{attribute 'linkalways'} 
{attribute 'no_explicit_call' := 'This FB is a CLASS and must be accessed using methods or properties'}
{attribute 'enable_dynamic_creation'}
FUNCTION_BLOCK _ETcWatchdogAccumulationType EXTENDS EnumDatatypeBase
VAR
	localData : ETcWatchdogAccumulationType;
	activeData : REFERENCE TO ETcWatchdogAccumulationType;
	enumBaseDatatype : _UINT(localData);
END_VAR

METHOD PRIVATE AddLocalEnumeration
VAR_INPUT
	Enumeration : T_MAXSTRING;
	Value : ETcWatchdogAccumulationType;
END_VAR
AddEnumeration(Enumeration, Value);
END_METHOD

PROPERTY PUBLIC Address : PVOID
GET
Address := ADR(activeData);
END_GET
END_PROPERTY

METHOD PUBLIC ClearReference
VAR_INPUT
END_VAR
activeData REF= localData;
SetBaseDatatypeReference();
END_METHOD

METHOD PUBLIC Clone : I_Datatype
VAR
    pClone : POINTER TO _ETcWatchdogAccumulationType;
END_VAR
pClone := __NEW(_ETcWatchdogAccumulationType(InitialValue := Value));
Clone := pClone^;
END_METHOD

METHOD FB_init : BOOL
VAR_INPUT
	bInitRetains : BOOL; // if TRUE, the retain variables are initialized (warm start / cold start)
	bInCopyCode : BOOL;  // if TRUE, the instance afterwards gets moved into the copy code (online change)
	InitialValue : ETcWatchdogAccumulationType;
END_VAR
localData := InitialValue;
AddBaseDatatype(enumBaseDatatype);
ClearReference();

AddLocalEnumeration('WD_ACC_TYPE_MEAN', ETcWatchdogAccumulationType.WD_ACC_TYPE_MEAN);
AddLocalEnumeration('WD_ACC_TYPE_PRODUCT', ETcWatchdogAccumulationType.WD_ACC_TYPE_PRODUCT);
END_METHOD

PROPERTY PUBLIC Identifier : T_MAXSTRING
GET
Identifier := 'ETcWatchdogAccumulationType';
END_GET
END_PROPERTY

METHOD IsEnumeratorValueEqual : BOOL
VAR_INPUT
	Enumerator : I_KeyValueForwardEnumerator;
END_VAR
VAR
	storedValue : ETcWatchdogAccumulationType;
END_VAR
IF NOT Enumerator.TryGet(storedValue) THEN
	RETURN;
END_IF

IsEnumeratorValueEqual := storedValue = activeData;
END_METHOD

METHOD PUBLIC MakeReferenceTo
VAR_INPUT
	ReferenceTarget : REFERENCE TO ETcWatchdogAccumulationType;
END_VAR
activeData REF= ReferenceTarget;
SetBaseDatatypeReference();
END_METHOD

METHOD PROTECTED SetBaseDatatypeReference
VAR_INPUT
END_VAR
enumBaseDatatype.MakeReferenceTo(activeData);
END_METHOD

PROPERTY PUBLIC Size : UDINT
GET
Size := SIZEOF(activeData);
END_GET
END_PROPERTY

METHOD TryMakeReferenceTo : BOOL
VAR_INPUT
	Target : I_Datatype;
END_VAR
VAR
	targetAsEnum : I_EnumDatatype;
	pTargetData : POINTER TO ETcWatchdogAccumulationType;
END_VAR
IF NOT Target.TryResolveAsEnumDatatype(targetAsEnum) THEN
	RETURN;
END_IF

IF targetAsEnum.Identifier <> Identifier THEN
	RETURN;
END_IF

pTargetData := Target.Address;
activeData REF= pTargetData^;
SetBaseDatatypeReference();
TryMakeReferenceTo := TRUE;
END_METHOD

PROPERTY PUBLIC Value : ETcWatchdogAccumulationType
GET
Value := activeData;
END_GET
SET
activeData := Value;
END_SET
END_PROPERTY

END_FUNCTION_BLOCK

(* stored: Version 1.1.0.1
   POU _ETcWatchdogAccumulationType: Id {9f8e712b-221d-4b7e-b23d-5a6a9598707e}, SpecialFunc None
   Folder Constructor: Id {27fa2eca-7872-442a-902d-23232a8fd823}
   Folder Private: Id {269bf6d6-2bb1-4317-9a0b-7ba3ebc69cf2}
   Folder Protected: Id {27d71b63-69c6-4680-925a-32c6207d271a}
   Method AddLocalEnumeration: Id {07002d06-a67f-4aba-b328-3283cf7e4720}
   Property Address: Id {1f239f12-6e32-4dcd-ab6c-6a0ce4ef1111}
   Get Get: Id {4769a909-79a9-470c-ae4f-3b56ce2ea6f9}
   Method ClearReference: Id {28bdb0ed-da8b-44d6-9f97-70731fff0c14}
   Method Clone: Id {6c808ac7-8fbb-4052-95bd-8df91069ec9b}
   Method FB_init: Id {634ef7f5-6f96-4ba5-b9a9-01fa2cf31a10}
   Property Identifier: Id {0ffe4e56-f1d2-4d1c-8de7-916a00535246}
   Get Get: Id {2633fb2b-a053-4228-b875-a7050c1535ff}
   Method IsEnumeratorValueEqual: Id {f02bc429-b086-42d4-b511-c7b98a1c12ff}
   Method MakeReferenceTo: Id {6e05ed69-6db9-4733-b551-c0c1f5e812dc}
   Method SetBaseDatatypeReference: Id {e6be49f2-20bf-4f80-ba26-a001d5b35436}
   Property Size: Id {19e13549-991c-4aa7-9d39-466cda80e336}
   Get Get: Id {bc022000-e4f6-4bae-8e46-482217014613}
   Method TryMakeReferenceTo: Id {12b1ec98-d1e3-48e8-b968-f53f969e7356}
   Property Value: Id {34a5055c-b9da-4aa6-8f2f-edc15276c009}
   Get Get: Id {a9f487fe-cf99-48d1-b1b3-acf3b7106997}
   Set Set: Id {8c31b69b-f31e-4874-99fc-2d889e00f01f} *)
